TYPE TcaTrolleyService :
STRUCT

END_STRUCT
END_TYPE

(* stored: Version 1.1.0.1
   DUT TcaTrolleyService: Id {2bac8508-f511-42e9-9c54-e2afb1919f2e} *)
